{attribute 'qualified_only'}
TYPE ENUM_LIC_States :
(
    Unknown := 0,
    OUT := 1,
    MIRROR1 := 2,
    MIRROR2 := 3,
    TARGET := 4
);
END_TYPE

(* stored: Version 1.1.0.1
   DUT ENUM_LIC_States: Id {c8ed19bc-c7b4-45d8-a75f-020a0ed98bf8} *)
